// TIA Portal V19 export
FUNCTION_BLOCK "FB80_TeepTrack"   // FB80, LAD
{ S7_Optimized_Access := 'TRUE' }
// stored: AutoNumber false, MemoryReserve 100, SetENOAutomatically false
   VAR_INPUT
      xProdRunning { ExternalAccessible := 'False'; ExternalVisible := 'False'; ExternalWritable := 'False'} : Bool;   // Production Running
      tTimePulse { ExternalAccessible := 'False'; ExternalVisible := 'False'; ExternalWritable := 'False'} : Time;   // Time for pulse StartStop
   END_VAR
   VAR_OUTPUT
      xPulseStartStop { ExternalAccessible := 'False'; ExternalVisible := 'False'; ExternalWritable := 'False'} : Bool;   // Pulse Start stop
      xRunProd { ExternalAccessible := 'False'; ExternalVisible := 'False'; ExternalWritable := 'False'} : Bool;   // Production running
   END_VAR
   VAR
      sxMemRun { ExternalAccessible := 'False'; ExternalVisible := 'False'; ExternalWritable := 'False'} : Bool;
      miDB_PulseStartStop { ExternalAccessible := 'False'; ExternalVisible := 'False'; ExternalWritable := 'False'; S7_SetPoint := 'True'} : TP_TIME;
      sxFPMemRun { ExternalAccessible := 'False'; ExternalVisible := 'False'; ExternalWritable := 'False'} : Bool;
      sxFNMemRun { ExternalAccessible := 'False'; ExternalVisible := 'False'; ExternalWritable := 'False'} : Bool;
   END_VAR
   VAR_TEMP   // added for the SCL form of the ladder/FBD networks
      _w1 : Bool;
      _w2 : Bool;
   END_VAR
BEGIN

REGION Network 1: Production running
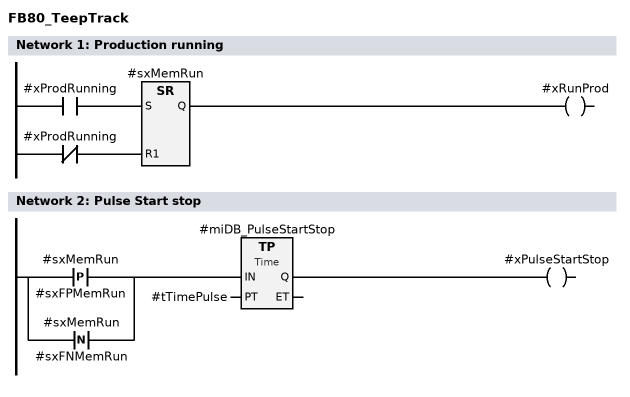
   RUNG wire#powerrail
      Contact( #xProdRunning )
      S_SR(operand := #sxMemRun, r1 := wire#w1)
      Coil( #xRunProd )
   END_RUNG
   RUNG wire#powerrail
      I_Contact( #xProdRunning )
   END_RUNG wire#w1
   // the same network as SCL:
   IF #xProdRunning THEN
       #sxMemRun := TRUE;   // SR flip-flop
   END_IF;
   IF NOT #xProdRunning THEN #sxMemRun := FALSE; END_IF;
   #xRunProd := #sxMemRun;
END_REGION

REGION Network 2: Pulse Start stop
   RUNG wire#powerrail
      P_Contact(operand := #sxMemRun, bit := #sxFPMemRun)
      wire#w1
      { S7_Templates := "time_type := Time" } #miDB_PulseStartStop.TP(pt := #tTimePulse, et =>)
      Coil( #xPulseStartStop )
   END_RUNG
   RUNG wire#powerrail
      N_Contact(operand := #sxMemRun, bit := #sxFNMemRun)
   END_RUNG wire#w1
   // the same network as SCL:
   #_w1 := #sxMemRun AND NOT #sxFPMemRun;   // rising edge of #sxMemRun
   #sxFPMemRun := #sxMemRun;
   #_w2 := NOT #sxMemRun AND #sxFNMemRun;   // falling edge of #sxMemRun
   #sxFNMemRun := #sxMemRun;
   #miDB_PulseStartStop(IN := #_w1 OR #_w2, PT := #tTimePulse);   // TP
   #xPulseStartStop := #miDB_PulseStartStop.Q;
END_REGION
END_FUNCTION_BLOCK
